(* IEC 61131-3 sources: ATCMcontrol_Engineering/src/TargetBase/Libs/ATCM_IEC1131_3/table_34, 2 files *)

(* ---- rs.st ---- *)
FUNCTION_BLOCK RS
VAR_INPUT
   S  : BOOL;
   R1 : BOOL;
END_VAR
VAR_OUTPUT
   Q1 : BOOL;
END_VAR

(*
 Q1 := NOT R1 AND (S OR Q1);
*)
inline { STDLIB(rs) }

END_FUNCTION_BLOCK

(* ---- sr.st ---- *)
FUNCTION_BLOCK SR
VAR_INPUT
   S1 : BOOL;
   R  : BOOL;
END_VAR
VAR_OUTPUT
   Q1 : BOOL;
END_VAR

(*
  Q1 := (NOT R AND Q1) OR S1;
*)
inline { STDLIB(SR) }

END_FUNCTION_BLOCK
